FUNCTION_BLOCK T_ComponentsResetClearsErrors EXTENDS T_UnitTestBase
VAR
  list : T_ComponentsCollection(10);
  newComponent, newComponent2 : T_ComponentMock; 
  actual1, actual2 : BOOL;
END_VAR

// Arrange
list.AddComponent(newComponent);
list.AddComponent(newComponent2);

//Act
list.CyclicLogic();
newComponent._error := TRUE;
newComponent2._error := TRUE;
list.Reset();

//Assert
actual1 := NOT newComponent.Error;
actual2 := NOT newComponent2.Error;
assertion.AssertEquals_BOOL(TRUE, actual1, 'actual1 := newComponent.Error;');
assertion.AssertEquals_BOOL(TRUE, actual2, 'actual2 := newComponent2.Error;');
TestFinished();

END_FUNCTION_BLOCK

(* stored: Version 1.1.0.1, ProductVersion 3.1.4024.12
   POU T_ComponentsResetClearsErrors: Id {1223cfde-ebb7-4b33-9c37-a9f533c9685d}, SpecialFunc None *)
